(* 计算某个日期 *)
FUNCTION calcDayNumber : dint
VAR_INPUT
	Year : DINT;
	Month : DINT;
	Day : DINT;
END_VAR
VAR
END_VAR

month := (month + 9) MOD 12;
year := year - month / 10;
calcDayNumber := (
        365 * year
        + year / 4
        - year / 100
        + year / 400
        + (month * 306 + 5) / 10
        + (day - 1)
    );

END_FUNCTION

(* stored: Version 1.1.0.1, ProductVersion 3.1.4024.12
   POU calcDayNumber: Id {a5b43f16-9a7f-41dd-9dd3-a9209260c24b}, SpecialFunc None *)
